# EPICS substitutions: lensApp/Db/monitor.substitutions
file monitor.tpl-db
{
    {
        LOCATION = $(LOCATION)
    }
}
